FUNCTION_BLOCK DATA_MERGE (* Basic Function Block Type *)
  (* Standard: 61499-2 *)
  (* Version 0.0, 12/28/2022, Dmitrii, Flexbridge AB, Template *)
  PACKAGE UAO.Hackathon;
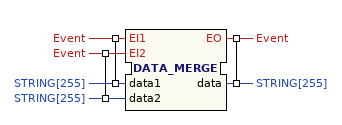
  EVENT_INPUT
    EI1 WITH data1; (* Normal Execution Request *)
    EI2 WITH data2;
  END_EVENT
  EVENT_OUTPUT
    EO WITH data; (* Execution Confirmation *)
  END_EVENT
  VAR_INPUT
    data1 : STRING[255]; (* Input event qualifier *)
    data2 : STRING[255];
  END_VAR
  VAR_OUTPUT
    data : STRING[255]; (* Output event qualifier *)
  END_VAR
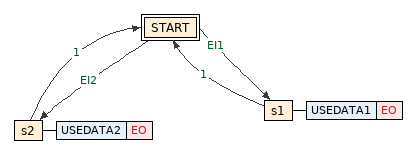
  EC_STATES
    START; (* Initial State *)
    s1 : USEDATA1 -> EO; (* Initialization *)
    s2 : USEDATA2 -> EO; (* Normal execution *)
  END_STATES
  EC_TRANSITIONS
    START TO s1 := EI1;
    s1 TO START := 1;
    START TO s2 := EI2;
    s2 TO START := 1;
  END_TRANSITIONS
  ALGORITHM USEDATA2 IN ST: (* Normally executed algorithm *)
;
data:=data2;
  END_ALGORITHM
  ALGORITHM USEDATA1 IN ST:
;
data:=data1;
  END_ALGORITHM
END_FUNCTION_BLOCK
